TYPE ST_P_SET_RECIPE :
STRUCT
	RecipeName:			STRING;
END_STRUCT
END_TYPE

(* stored: Version 1.1.0.1, ProductVersion 3.1.4024.10
   DUT ST_P_SET_RECIPE: Id {ade5b1da-1fcf-4ee9-9575-51004284275f} *)
